(* CODESYS project Test01.project

Project tree, tasks and I/O mapping:
  Device : Elmo Platinum Maestro, Elmo Motion Control, version 1.0.0.2
    application Application
      libraries: Standard, * (System)
      task MainTask (cyclic, interval t#20ms, priority 1) calls PLC_PRG
      program PLC_PRG [ST]
      function fCalculate [ST]
      function block fbCalculate [ST]
    Elmo_Master_Device : Elmo Master Device, Elmo, version 1.0.0.2
*)

// Device/Application/PLC_PRG
PROGRAM PLC_PRG
VAR CONSTANT
	c_uiObject : UINT := 10;
END_VAR
VAR
	iCnt: INT := 0;
	xBtn: BOOL;
	xLight: BOOL;
	uiStep: UINT;
	
	tonTimer1 : ton;
	xStart: BOOL;
	tTimer1: TIME:= T#100MS;
	
	//c_uiObject: UINT:=10;
	xState: ARRAY[1..c_uiObject] OF BOOL;
	uiLoop: UINT;
	
	fbCalc1 : fbCalculate;
END_VAR


//iCnt := iCnt + 5;
iCnt := fCalculate(ii_Cnt := iCnt);
(*
IF iCnt >=0 AND iCnt < 2000 THEN
	xLight := TRUE;
ELSIF iCnt >= 2000 AND iCnt<3000 THEN
	xLight:= FALSE;
ELSE
	iCnt:=0;
END_IF
*)

//xLight := fCalculate(iCnt);

(*
tonTimer1(IN := xStart, PT := tTimer1);
CASE uiStep OF
	10:
	(*
	   xStart := TRUE;
	   IF tonTimer1.Q THEN
		   xStart := FALSE;
		   uiStep:= 20;
	   END_IF
	   *)
	   FOR uiLoop:=1 TO c_uiObject BY 1 DO
		   xState[uiLoop] := TRUE;
	   END_FOR
	   uiStep:= 20;
	   
	20:
	   xStart := TRUE;
	   IF tonTimer1.Q THEN
		   xStart := FALSE;
		   uiStep:= 30;
	   END_IF
	30:
	(*
	   xStart := TRUE;
	   IF tonTimer1.Q THEN
		   xStart := FALSE;
		   uiStep:= 10;
	   END_IF
	   *)
	   FOR uiLoop:=1 TO c_uiObject BY 1 DO
		   xState[uiLoop] := FALSE;
	   END_FOR
	   uiStep:= 40;
	 40:
	   xStart := TRUE;
	   IF tonTimer1.Q THEN
		   xStart := FALSE;
		   uiStep:= 10;
	   END_IF
	ELSE
		uiStep:=10;
END_CASE


WHILE iCnt < 10 DO
	iCnt := iCnt + 1;
END_WHILE
*)

fbCalc1(ii_Cnt := iCnt, ox_Light => xLight);

END_PROGRAM

// Device/Application/fCalculate
FUNCTION fCalculate : int
VAR_INPUT
	ii_Cnt : INT;
END_VAR
VAR
END_VAR

IF ii_Cnt >=3000 THEN
	fCalculate := 0;
//ELSIF ii_Cnt >= 2000 AND ii_Cnt<3000 THEN
	//fCalculate:= FALSE;
ELSE
	fCalculate := ii_Cnt + 1;
END_IF

END_FUNCTION

// Device/Application/fbCalculate
FUNCTION_BLOCK fbCalculate
VAR_INPUT
	ii_Cnt : INT;
END_VAR
VAR_OUTPUT
	ox_Light : BOOL;
END_VAR
VAR
END_VAR

IF ii_Cnt >= 0 AND ii_cnt < 2000 THEN
	ox_Light := TRUE;
ELSIF ii_Cnt >= 2000 AND ii_Cnt < 3000 THEN
	ox_Light := FALSE;
END_IF

END_FUNCTION_BLOCK
